// TIA Portal V15 export
TextList "Textlist"  ListRange=Decimal
  TextListEntry   EntryType=SingleValue, Text="?"
